TYPE
    ST_BEPointDefinitions : STRUCT
        MinCarriagePos  : REAL;
        Infeed          : REAL;
        PrePress        : REAL;
        PostPress       : REAL;
        AssemblyHandoff : REAL;
        PickPoint_1     : REAL;
        MaxCarriagePos  : REAL;
    END_STRUCT
END_TYPE

(* stored: Version 1.1.0.1
   DUT ST_BEPointDefinitions: Id {a4e60e0e-6251-467e-bd37-a487a5441484} *)
